{attribute 'GeneratedUsingTerminal: EJ1914-0000-0017'}
{attribute addProperty BoxType "EJ1914-0000-0017"}
{attribute addProperty Id "Safe_Logic_StateAT %I*USINT1Cycle_CounterAT %I*USINT1"}
{attribute addProperty CRC "4008261774"}
{attribute addProperty Size "2"}
TYPE FSLOGIC_Inputs_EEE9388E :
STRUCT
	{attribute addProperty Name "Safe_Logic_State"}
	Safe_Logic_State AT %I* : USINT;
	{attribute addProperty Name "Cycle_Counter"}
	Cycle_Counter AT %I* : USINT;
END_STRUCT
END_TYPE

(* stored: Version 1.2.0.0, ProductVersion 3.1.4024.9
   DUT FSLOGIC_Inputs_EEE9388E: Id {4c867a45-4bd5-484e-b255-16968536b131} *)
